KUKA KRL program: MyProgram.src

&ACCESS RVP
&REL 9
&PARAM EDITMASK = *
&PARAM TEMPLATE = C:\KRC\Roboter\Template\vorgabe
DEF MyProgram()
; ***PROGRAM_GENERATED_BY_______***
; ***MW__________________***
; ***FOR_MELTIO_DIRECTEDMETAL3D_***

Un_init()
TOOL_DATA[3]={FRAME: X 252.94,Y 0.13,Z 196.30,A 0,B -89.92,C 0.07}
BASE_DATA[4]={FRAME: X 1499.49,Y 0.55,Z 394.19,A 0.0,B 0.15,C 0.03}

; FOLD Initialise and set default speed
BAS (#INITMOV,0)
BAS (#VEL_PTP,100)
BAS (#ACC_PTP,20)
;BAS (#TOOL,0)
;BAS (#BASE,0)
;ENDFOLD

$ADVANCE = 5

;onStart
$APO.CPTP = 1
$APO.CDIS = 1

; ---- Setting reference (Base) ----
$BASE = BASE_DATA[4]
; --------------------------

; ---- Setting tool (TCP) ----
$TOOL = TOOL_DATA[3]
; --------------------------
VEL_APROX_PRINT=0.04
VEL_PRINT=0.01
DELAY_PROCESS_ON=5
VEL_DTIME=15
; Stage Two Robot Integration Simplified
$VEL.CP = 0.05
PTP $POS_ACT
LIN {E6POS: X 0.000,Y 0.000,Z 200.000,A 0,B 0,C 0,E1 0,E2 -45.0} C_DIS

;FOLD PRINT START
ENABLE_PROCESS = TRUE; Print Enable Status
WAIT SEC DELAY_PROCESS_ON;
;ENDFOLD Delay process

InitDeposition();
MyProgram_000()
MyProgram_001()
MyProgram_002()
MyProgram_003()
MyProgram_004()
MyProgram_005()
MyProgram_006()
MyProgram_007()
MyProgram_008()
MyProgram_009()
MyProgram_010()
MyProgram_011()
MyProgram_012()
MyProgram_013()
MyProgram_014()
MyProgram_015()
MyProgram_016()
MyProgram_017()
MyProgram_018()
MyProgram_019()
MyProgram_020()
MyProgram_021()
MyProgram_022()
MyProgram_023()
MyProgram_024()
MyProgram_025()
MyProgram_026()
MyProgram_027()
MyProgram_028()
MyProgram_029()
MyProgram_030()
MyProgram_031()
MyProgram_032()
MyProgram_033()
MyProgram_034()
MyProgram_035()
MyProgram_036()
MyProgram_037()
MyProgram_038()
MyProgram_039()
MyProgram_040()
MyProgram_041()
MyProgram_042()
MyProgram_043()
MyProgram_044()
MyProgram_045()
MyProgram_046()
MyProgram_047()
MyProgram_048()
MyProgram_049()
MyProgram_050()
MyProgram_051()
MyProgram_052()
MyProgram_053()
MyProgram_054()
MyProgram_055()
MyProgram_056()
MyProgram_057()
MyProgram_058()
MyProgram_059()
MyProgram_060()
MyProgram_061()
MyProgram_062()
MyProgram_063()
MyProgram_064()
MyProgram_065()
MyProgram_066()
MyProgram_067()
MyProgram_068()
MyProgram_069()
MyProgram_070()
MyProgram_071()
MyProgram_072()
MyProgram_073()
MyProgram_074()
MyProgram_075()
MyProgram_076()
MyProgram_077()
MyProgram_078()
MyProgram_079()
MyProgram_080()
MyProgram_081()
MyProgram_082()
MyProgram_083()
MyProgram_084()
MyProgram_085()
MyProgram_086()
MyProgram_087()
MyProgram_088()
MyProgram_089()
MyProgram_090()
MyProgram_091()
MyProgram_092()
MyProgram_093()
MyProgram_094()
MyProgram_095()
MyProgram_096()
MyProgram_097()
MyProgram_098()
MyProgram_099()
MyProgram_100()
MyProgram_101()
MyProgram_102()
MyProgram_103()
MyProgram_104()
MyProgram_105()
MyProgram_106()
MyProgram_107()
MyProgram_108()
MyProgram_109()
MyProgram_110()
MyProgram_111()
MyProgram_112()
MyProgram_113()
MyProgram_114()
MyProgram_115()
MyProgram_116()
MyProgram_117()
MyProgram_118()
MyProgram_119()
MyProgram_120()
MyProgram_121()
MyProgram_122()
MyProgram_123()
MyProgram_124()
MyProgram_125()
MyProgram_126()
MyProgram_127()
MyProgram_128()
MyProgram_129()
MyProgram_130()
MyProgram_131()
MyProgram_132()
MyProgram_133()
MyProgram_134()
MyProgram_135()
MyProgram_136()
MyProgram_137()
MyProgram_138()
MyProgram_139()
MyProgram_140()
MyProgram_141()
MyProgram_142()
MyProgram_143()
MyProgram_144()
MyProgram_145()
MyProgram_146()
MyProgram_147()
MyProgram_148()
MyProgram_149()
MyProgram_150()
MyProgram_151()
MyProgram_152()
MyProgram_153()
MyProgram_154()
MyProgram_155()
MyProgram_156()
MyProgram_157()
MyProgram_158()
MyProgram_159()
MyProgram_160()
MyProgram_161()
MyProgram_162()
MyProgram_163()
MyProgram_164()
MyProgram_165()
MyProgram_166()
MyProgram_167()
MyProgram_168()
MyProgram_169()
MyProgram_170()
MyProgram_171()
MyProgram_172()
MyProgram_173()
MyProgram_174()
MyProgram_175()
MyProgram_176()
MyProgram_177()
MyProgram_178()
MyProgram_179()
MyProgram_180()
MyProgram_181()
MyProgram_182()
MyProgram_183()
MyProgram_184()
MyProgram_185()
MyProgram_186()
MyProgram_187()
MyProgram_188()
MyProgram_189()
MyProgram_190()
MyProgram_191()
MyProgram_192()
MyProgram_193()
MyProgram_194()
MyProgram_195()
MyProgram_196()
MyProgram_197()
MyProgram_198()
MyProgram_199()
MyProgram_200()
MyProgram_201()
MyProgram_202()
MyProgram_203()
MyProgram_204()
MyProgram_205()
MyProgram_206()
MyProgram_207()
MyProgram_208()
MyProgram_209()
MyProgram_210()
MyProgram_211()
MyProgram_212()
MyProgram_213()
MyProgram_214()
MyProgram_215()
MyProgram_216()
MyProgram_217()
MyProgram_218()
MyProgram_219()
MyProgram_220()
MyProgram_221()
MyProgram_222()
MyProgram_223()
MyProgram_224()
MyProgram_225()
MyProgram_226()
MyProgram_227()
MyProgram_228()
MyProgram_229()
MyProgram_230()
MyProgram_231()
MyProgram_232()
MyProgram_233()
MyProgram_234()
MyProgram_235()
MyProgram_236()
MyProgram_237()
MyProgram_238()
MyProgram_239()
MyProgram_240()
MyProgram_241()
MyProgram_242()
MyProgram_243()
MyProgram_244()
MyProgram_245()
MyProgram_246()
MyProgram_247()
MyProgram_248()
MyProgram_249()
MyProgram_250()
MyProgram_251()
MyProgram_252()
MyProgram_253()
MyProgram_254()
MyProgram_255()
MyProgram_256()
MyProgram_257()
MyProgram_258()
MyProgram_259()
MyProgram_260()
MyProgram_261()
MyProgram_262()
MyProgram_263()
MyProgram_264()
MyProgram_265()
MyProgram_266()
MyProgram_267()
MyProgram_268()
MyProgram_269()
MyProgram_270()
MyProgram_271()
MyProgram_272()
MyProgram_273()
MyProgram_274()
MyProgram_275()
MyProgram_276()
MyProgram_277()
MyProgram_278()
MyProgram_279()
MyProgram_280()
MyProgram_281()
MyProgram_282()
MyProgram_283()
MyProgram_284()
MyProgram_285()
MyProgram_286()
MyProgram_287()
MyProgram_288()
MyProgram_289()
MyProgram_290()
MyProgram_291()
MyProgram_292()
MyProgram_293()
MyProgram_294()
MyProgram_295()
MyProgram_296()
MyProgram_297()
MyProgram_298()
MyProgram_299()
MyProgram_300()
MyProgram_301()
MyProgram_302()
MyProgram_303()
MyProgram_304()
MyProgram_305()
MyProgram_306()
MyProgram_307()
MyProgram_308()
MyProgram_309()
MyProgram_310()
MyProgram_311()
MyProgram_312()
MyProgram_313()
MyProgram_314()
MyProgram_315()
MyProgram_316()
MyProgram_317()
MyProgram_318()
MyProgram_319()
MyProgram_320()
MyProgram_321()
MyProgram_322()
MyProgram_323()
MyProgram_324()
MyProgram_325()
MyProgram_326()
MyProgram_327()
MyProgram_328()
MyProgram_329()
MyProgram_330()
MyProgram_331()
MyProgram_332()
MyProgram_333()
MyProgram_334()
MyProgram_335()
MyProgram_336()
MyProgram_337()
MyProgram_338()
MyProgram_339()
MyProgram_340()
MyProgram_341()
MyProgram_342()
MyProgram_343()
MyProgram_344()
MyProgram_345()
ResetDeposition();
PTP $POS_ACT

END
